FUNCTION_BLOCK BufferingProduct EXTENDS BaseState
VAR_INPUT
END_VAR
VAR_OUTPUT
END_VAR
VAR
	InternalBufferingTime : TIME;
END_VAR

METHOD mIrun : BOOL
IF BasePointer^.ProximityAccessI[1].mReturnBOOL() THEN;
	IF mCheckDosing() THEN
		StateTimer(IN:= TRUE, PT:=InternalBufferingTime);
		IF StateTimer.Q = TRUE THEN
			mNextState();
			StateTimer(IN:= FALSE);
//		ELSE
//			RETURN;
		END_IF
	END_IF
END_IF
END_METHOD

METHOD mStateInit : BOOL
VAR_INPUT
	BufferingTime : TIME;
END_VAR
InternalBufferingTime := BufferingTime;
END_METHOD

END_FUNCTION_BLOCK

(* stored: Version 1.1.0.1, ProductVersion 3.1.4024.12
   POU BufferingProduct: Id {8d0817e2-d07d-421a-bf5d-fec26434d4cc}, SpecialFunc None
   Method mIrun: Id {c0be4efb-a317-4090-b5d3-b2693ed7b2fa}
   Method mStateInit: Id {af1c1d9c-0dfe-461d-9f63-9f99d82bfff5} *)
